PROGRAM MAIN
VAR
	// 
	

	//----------------------------------------------------------------------oldschoo1
END_VAR

(* 	for Jabil, Bray @ Tegan Innovations, Waterford - July2025. Ireland
 	m/c TE1096-04 SISS _rev1.0
	>> design by oldschoo1
	>> smac and hmi by seb	*)

 
// Calling:
A_Master();
   A_HMI();
D_FaultHandling(); 
   
//Get System Time
//PRG_SysTime();
PRG_MasterSystemTime();
//--------------------------------------------------------------------------oldschoo1

END_PROGRAM

(* stored: Version 1.1.0.1, ProductVersion 3.1.4024.12
   POU MAIN: Id {e7fb6707-82b6-4a45-b743-0b2a74a45279}, SpecialFunc None *)
